FUNCTION RemoveStringFromEnd : T_MaxString
VAR_INPUT
	text : T_MaxString;
	end : T_MaxString;
END_VAR
VAR
	diff : INT;
END_VAR

diff := LEN(text) - LEN(end);
IF (diff < 0) THEN
	RemoveStringFromEnd := text;
	RETURN;
END_IF

IF (StringEndsWithAny(text, end)) THEN
	RemoveStringFromEnd := LEFT(text, diff);
END_IF

END_FUNCTION

(* stored: Version 1.1.0.1
   POU RemoveStringFromEnd: Id {a8d4f214-210e-0ce9-085f-79a2833122eb}, SpecialFunc None *)
